FUNCTION_BLOCK AUTOMATIC_SCREWING
VAR_INPUT
END_VAR
VAR_OUTPUT
END_VAR
VAR
END_VAR

ACTION ACT_SEQUENCE_CHAIN:
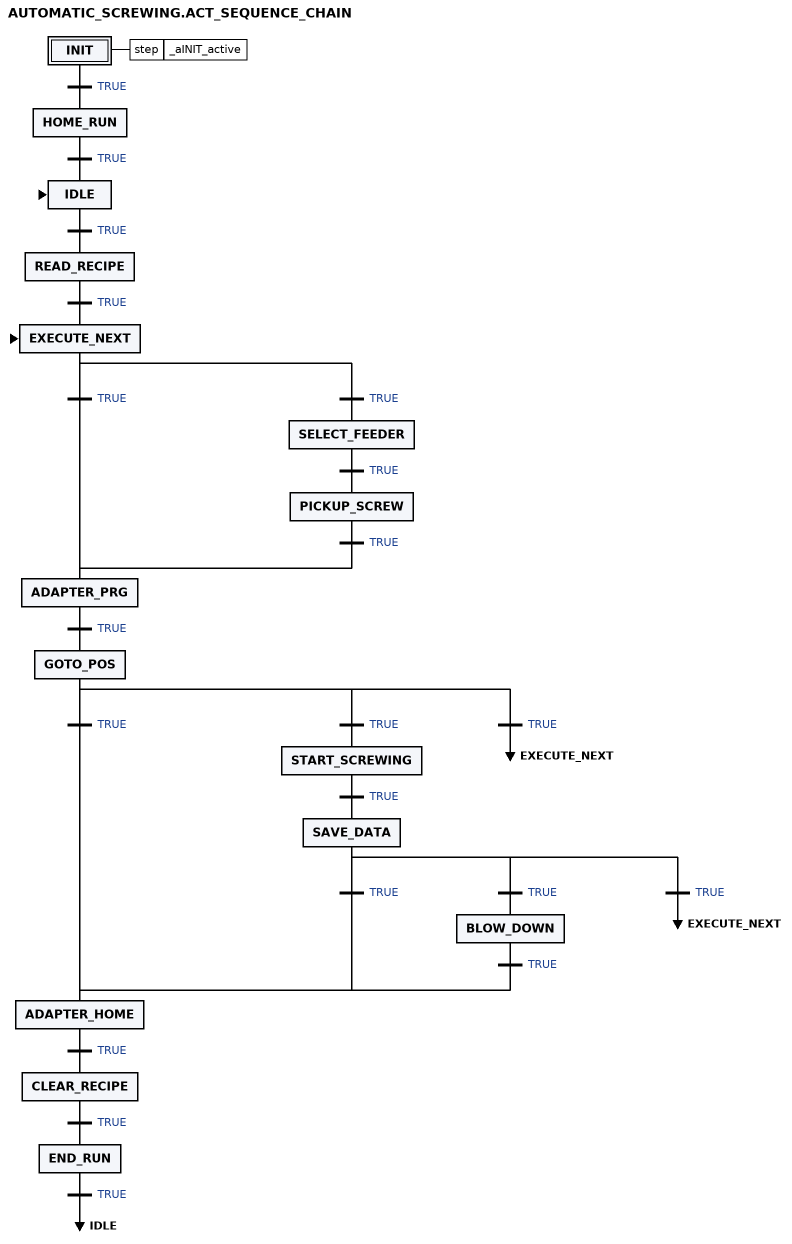
INITIAL_STEP INIT:
    _aINIT_active(N);  // step action
END_STEP
TRANSITION FROM INIT TO HOME_RUN
    := TRUE;
END_TRANSITION
STEP HOME_RUN:
END_STEP
TRANSITION FROM HOME_RUN TO IDLE
    := TRUE;
END_TRANSITION
STEP IDLE:
END_STEP
TRANSITION FROM IDLE TO READ_RECIPE
    := TRUE;
END_TRANSITION
STEP READ_RECIPE:
END_STEP
TRANSITION FROM READ_RECIPE TO EXECUTE_NEXT
    := TRUE;
END_TRANSITION
STEP EXECUTE_NEXT:
END_STEP
TRANSITION FROM EXECUTE_NEXT TO ADAPTER_PRG
    := TRUE;
END_TRANSITION
TRANSITION FROM EXECUTE_NEXT TO SELECT_FEEDER
    := TRUE;
END_TRANSITION
STEP SELECT_FEEDER:
END_STEP
TRANSITION FROM SELECT_FEEDER TO PICKUP_SCREW
    := TRUE;
END_TRANSITION
STEP PICKUP_SCREW:
END_STEP
TRANSITION FROM PICKUP_SCREW TO ADAPTER_PRG
    := TRUE;
END_TRANSITION
STEP ADAPTER_PRG:
END_STEP
TRANSITION FROM ADAPTER_PRG TO GOTO_POS
    := TRUE;
END_TRANSITION
STEP GOTO_POS:
END_STEP
TRANSITION FROM GOTO_POS TO ADAPTER_HOME
    := TRUE;
END_TRANSITION
TRANSITION FROM GOTO_POS TO START_SCREWING
    := TRUE;
END_TRANSITION
STEP START_SCREWING:
END_STEP
TRANSITION FROM START_SCREWING TO SAVE_DATA
    := TRUE;
END_TRANSITION
STEP SAVE_DATA:
END_STEP
TRANSITION FROM SAVE_DATA TO ADAPTER_HOME
    := TRUE;
END_TRANSITION
TRANSITION FROM SAVE_DATA TO BLOW_DOWN
    := TRUE;
END_TRANSITION
STEP BLOW_DOWN:
END_STEP
TRANSITION FROM BLOW_DOWN TO ADAPTER_HOME
    := TRUE;
END_TRANSITION
TRANSITION FROM SAVE_DATA TO EXECUTE_NEXT
    := TRUE;
END_TRANSITION
TRANSITION FROM GOTO_POS TO EXECUTE_NEXT
    := TRUE;
END_TRANSITION
STEP ADAPTER_HOME:
END_STEP
TRANSITION FROM ADAPTER_HOME TO CLEAR_RECIPE
    := TRUE;
END_TRANSITION
STEP CLEAR_RECIPE:
END_STEP
TRANSITION FROM CLEAR_RECIPE TO END_RUN
    := TRUE;
END_TRANSITION
STEP END_RUN:
END_STEP
TRANSITION FROM END_RUN TO IDLE
    := TRUE;
END_TRANSITION
// branch label Branch2_ACT_SEQUENCE_CHAIN
// branch label Branch3_ACT_SEQUENCE_CHAIN
// branch label Branch0_ACT_SEQUENCE_CHAIN
END_ACTION

END_FUNCTION_BLOCK

(* stored: Version 1.1.0.1, ProductVersion 3.1.4022.18
   POU AUTOMATIC_SCREWING: Id {4784e865-14ee-4869-804b-679825818e9e}, SpecialFunc None
   Action ACT_SEQUENCE_CHAIN: Id {3d9a410c-3808-4c2d-9504-cdfa3b5d8e53} *)
